FUNCTION Buffer_Layout_Set_Real_Array : UINT
VAR_INPUT
END_VAR
VAR
END_VAR

END_FUNCTION

(* stored: Version 1.1.0.1, ProductVersion 3.1.4024.10
   POU Buffer_Layout_Set_Real_Array: Id {aca91fad-8d84-4aab-a074-7d2f874df1de}, SpecialFunc None *)
